// TIA Portal V16 export
// export: Created 2021-04-06T19:52:19.7607963Z, ExportSetting WithDefaults, DisplayName Totally Integrated Automation Portal, DisplayVersion V16, DisplayName TIA Portal Version Control Interface, DisplayVersion V16, DisplayName TIA Portal Openness, DisplayVersion V16, DisplayName STEP 7 Professional, DisplayVersion V16, DisplayName STEP 7 Safety, DisplayVersion V16, DisplayName WinCC Unified SCADA Engineering System, DisplayVersion V16
TYPE "sourceConv"
// stored: IsFailsafeCompliant false
   STRUCT
      currentSpeed : Int;   // ОС скорость
      manSetSpeed : Int;   // ручн - задание скорости
      isConvWork : Bool;   // конв работает
      isConvAlarm : Bool;   // авария конв
      manStartConv : Bool;   // ручн - старт конвейера
      stateConvInt : Int;   // состояние конвейера
      setSpeedWeightLimit : Int;   // скорость питателя при перевесе
   END_STRUCT;
END_TYPE
